(* Logix 5000 project; controller cal1632 1756-L62 rev 16.20; software revision 16.05; part 59 of 61 *)
(* tags used below, declared in another part *)
   AFI : BOOL;
   FAULT : BOOL;
   HMI : BOOL;
   p00_lin_timer_pre_0ms : DINT;
   p00_lin_timer_pre_1s : DINT;
   p00_lin_timer_pre_disc : DINT;
   p00_wac : Accumulator;   // Winder Accumulator
   p01_param_master_decel : REAL;
   p01r09 : routine;
   p01r09_pb_global_reset : BOOL;
   p01r12_master_ramped_speed : REAL;
   p01r13_line_running : BOOL;
   p01r13_line_slow_ramp : BOOL;
   p02_recipe_from_hmi : recipe;
   p29_di_wdr_a : BOOL;
   p29_param_acc_park_sp : REAL;   // Winder Accumulator Speed Trim Park Setpoint - Where the Carriage Sits [% of Stroke]
   p29r09_torque_mode : BOOL;
   p29r09_winder_a_active : BOOL;
   p29r09_winder_b_active : BOOL;
   p29r10 : routine;
   p29r10_request_run : BOOL;
   p29r11 : routine;
   p29r11_request_run : BOOL;
   p29r15_request_run : BOOL;
   p29r16_request_run : BOOL;
   p30_di_pin_1 : BOOL;
   p30_di_pin_2 : BOOL;
   p30_di_pin_3 : BOOL;
   p30_di_pin_4 : BOOL;
   p30_di_pin_5 : BOOL;
   p30_di_pin_6 : BOOL;
   p30_di_pin_7 : BOOL;
   p30_di_pin_8 : BOOL;
   p30_di_retraction_down_ls : BOOL;
   p30_di_retraction_up_ls : BOOL;
   p30_di_rotation_fault : BOOL;
   p30_do_retract_motion : BOOL;
   p30_do_rotation_fwd : BOOL;
   p30_do_rotation_rev : BOOL;
   p30r09_mode_close : BOOL;
   p30r09_mode_open : BOOL;
   p30r10 : routine;
   p30r10_motion_monitor_dwell : TIMER;
   p30r10_request_close : BOOL;
   p30r10_request_monitor : BOOL;
   p30r10_request_open : BOOL;
   p30r10_run_permissive : BOOL;
   p30r10_safety_pins_stowed : BOOL;
   p30r10_timer_fault : TIMER[4];
   p30r10_timer_warning : TIMER[4];
(* P30_Retraction_System, continued *)

ROUTINE R10_Retraction   (* ladder *)
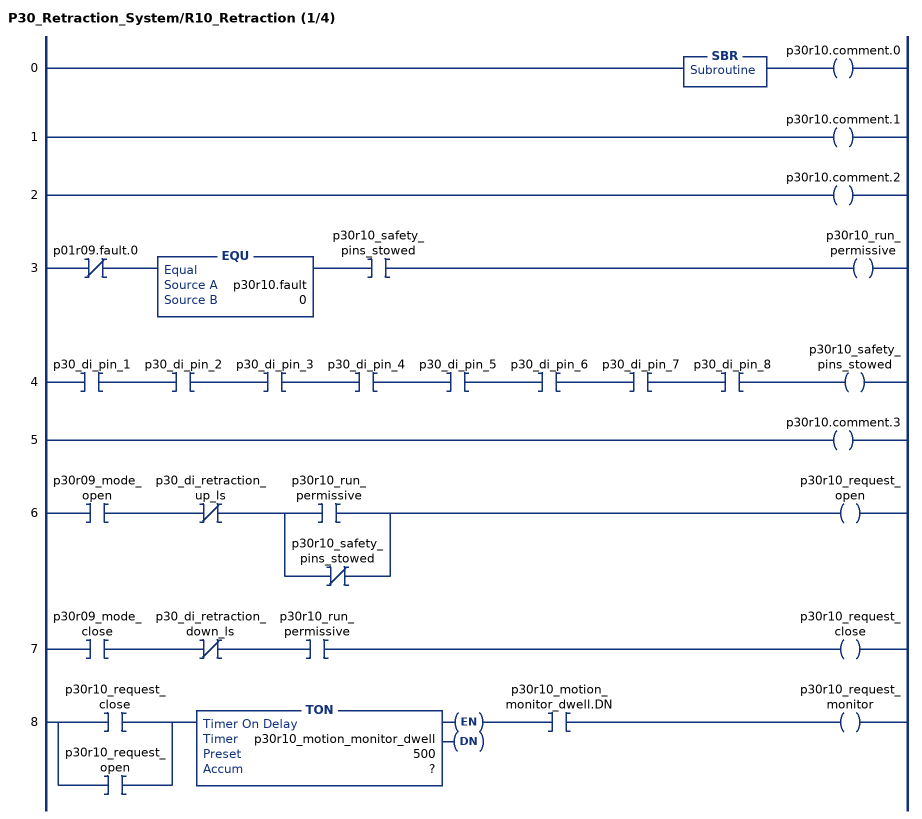
   0: SBR()OTE(p30r10.comment.0);
   1: OTE(p30r10.comment.1);
   2: OTE(p30r10.comment.2);
   3: XIO(p01r09.fault.0)EQU(p30r10.fault,0)XIC(p30r10_safety_pins_stowed)OTE(p30r10_run_permissive);
   4: XIC(p30_di_pin_1)XIC(p30_di_pin_2)XIC(p30_di_pin_3)XIC(p30_di_pin_4)XIC(p30_di_pin_5)XIC(p30_di_pin_6)XIC(p30_di_pin_7)XIC(p30_di_pin_8)OTE(p30r10_safety_pins_stowed);
   5: OTE(p30r10.comment.3);
   6: XIC(p30r09_mode_open)XIO(p30_di_retraction_up_ls)[XIC(p30r10_run_permissive) ,XIO(p30r10_safety_pins_stowed) ]OTE(p30r10_request_open);
   7: XIC(p30r09_mode_close)XIO(p30_di_retraction_down_ls)XIC(p30r10_run_permissive)OTE(p30r10_request_close);
   8: [XIC(p30r10_request_close) ,XIC(p30r10_request_open) ]TON(p30r10_motion_monitor_dwell,?,?)XIC(p30r10_motion_monitor_dwell.DN)OTE(p30r10_request_monitor);
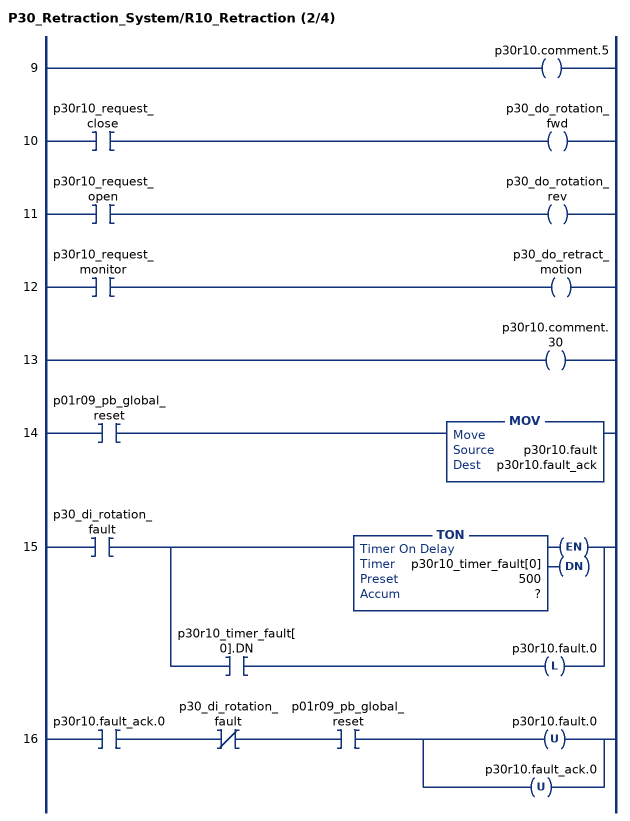
   9: OTE(p30r10.comment.5);
   10: XIC(p30r10_request_close)OTE(p30_do_rotation_fwd);
   11: XIC(p30r10_request_open)OTE(p30_do_rotation_rev);
   12: XIC(p30r10_request_monitor)OTE(p30_do_retract_motion);
   13: OTE(p30r10.comment.30);
   14: XIC(p01r09_pb_global_reset)MOV(p30r10.fault,p30r10.fault_ack);
   15: XIC(p30_di_rotation_fault)[TON(p30r10_timer_fault[0],?,?) ,XIC(p30r10_timer_fault[0].DN) OTL(p30r10.fault.0) ];
   16: XIC(p30r10.fault_ack.0)XIO(p30_di_rotation_fault)XIC(p01r09_pb_global_reset)[OTU(p30r10.fault.0) ,OTU(p30r10.fault_ack.0) ];
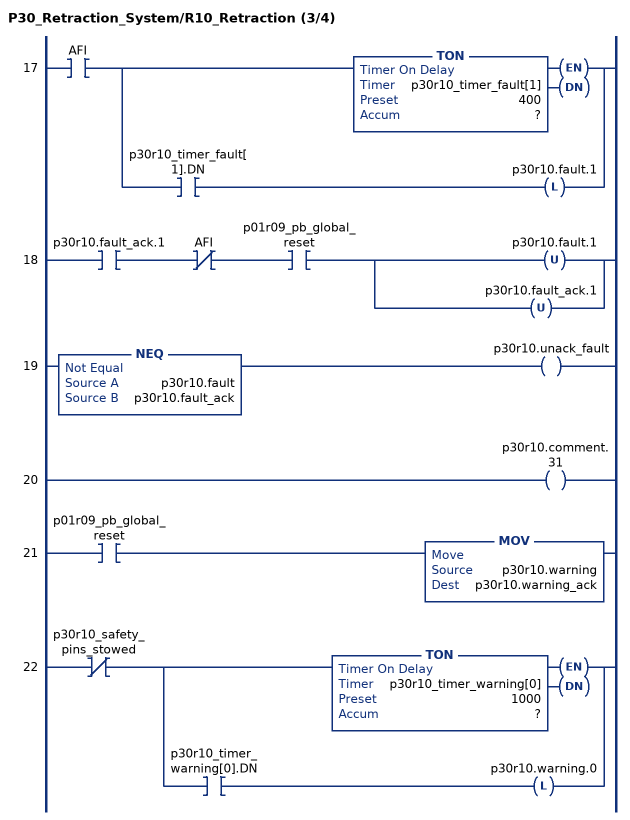
   17: XIC(AFI)[TON(p30r10_timer_fault[1],?,?) ,XIC(p30r10_timer_fault[1].DN) OTL(p30r10.fault.1) ];
   18: XIC(p30r10.fault_ack.1)XIO(AFI)XIC(p01r09_pb_global_reset)[OTU(p30r10.fault.1) ,OTU(p30r10.fault_ack.1) ];
   19: NEQ(p30r10.fault,p30r10.fault_ack)OTE(p30r10.unack_fault);
   20: OTE(p30r10.comment.31);
   21: XIC(p01r09_pb_global_reset)MOV(p30r10.warning,p30r10.warning_ack);
   22: XIO(p30r10_safety_pins_stowed)[TON(p30r10_timer_warning[0],?,?) ,XIC(p30r10_timer_warning[0].DN) OTL(p30r10.warning.0) ];
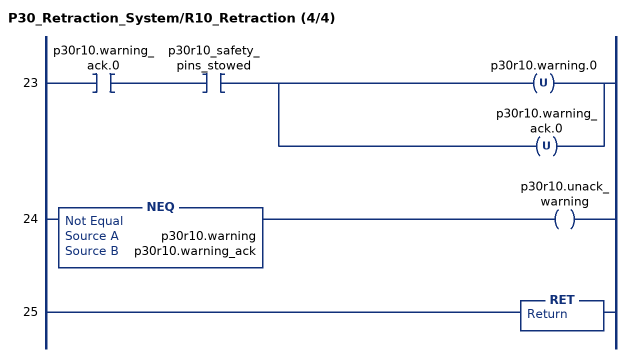
   23: XIC(p30r10.warning_ack.0)XIC(p30r10_safety_pins_stowed)[OTU(p30r10.warning.0) ,OTU(p30r10.warning_ack.0) ];
   24: NEQ(p30r10.warning,p30r10.warning_ack)OTE(p30r10.unack_warning);
   25: RET();
END_ROUTINE
END_PROGRAM

PROGRAM P31_WAC
// Winder Accumulator
VAR
   A00 : ALIAS FOR hmi_dint[0].0;
   A01 : ALIAS FOR hmi_dint[0].1;
   A02 : ALIAS FOR hmi_dint[0].2;
   A03 : ALIAS FOR hmi_dint[0].3;
   A04 : ALIAS FOR hmi_dint[0].4;
   A05 : ALIAS FOR hmi_dint[0].5;
   A06 : ALIAS FOR hmi_dint[0].6;
   A07 : ALIAS FOR hmi_dint[0].7;
   A08 : ALIAS FOR hmi_dint[0].8;
   A09 : ALIAS FOR hmi_dint[0].9;
   A10 : ALIAS FOR hmi_dint[0].10;
   A11 : ALIAS FOR hmi_dint[0].11;
   A12 : ALIAS FOR hmi_dint[0].12;
   A13 : ALIAS FOR hmi_dint[0].13;
   A14 : ALIAS FOR hmi_dint[0].14;
   A15 : ALIAS FOR hmi_dint[0].15;
   A16 : ALIAS FOR hmi_dint[0].16;
   A17 : ALIAS FOR hmi_dint[0].17;
   A18 : ALIAS FOR hmi_dint[0].18;
   A19 : ALIAS FOR hmi_dint[0].19;
   A20 : ALIAS FOR hmi_dint[0].20;
   A21 : ALIAS FOR hmi_dint[0].21;
   A22 : ALIAS FOR hmi_dint[0].22;
   A23 : ALIAS FOR hmi_dint[0].23;
   A24 : ALIAS FOR hmi_dint[0].24;
   A25 : ALIAS FOR hmi_dint[0].25;
   A26 : ALIAS FOR hmi_dint[0].26;
   A27 : ALIAS FOR hmi_dint[0].27;
   A28 : ALIAS FOR hmi_dint[0].28;
   A29 : ALIAS FOR hmi_dint[0].29;
   A30 : ALIAS FOR hmi_dint[0].30;
   A31 : ALIAS FOR hmi_dint[0].31;
   aaa_cjj_test_real1 : REAL;
   aaa_close_nip_from_feedroll : BOOL;
   acc_decel_reserve_pct : REAL;   // Accumulator Stroke Reserved for the Line Decel at the Present Line Speed [% of Stroke]
   acc_empty_limit : BOOL := 1;   // Accumulator Empty Limit
   acc_fill_status : DINT;
   acc_full_limit : BOOL;   // Accumulator Full Limit
   acc_norm_stop_pct : REAL := 60.0;   // Accumulator Normal Stop Threshold Computed - Full Limit Less Decel Reserve [% of Stroke]
   acc_position_last : REAL;
   acc_status : ALIAS FOR hmi_dint[13];
   accum_filling_on : ALIAS FOR hmi_dint[9].12;
   accum_holding_pressure_on : BOOL;   // Accumulator Holding Pressure Active
   accum_tension_pressure_on : BOOL := 1;   // Accumulator Tension Pressure Active
   accumulator_state : DINT := 33;   // Accumulator Sequence State Word
        .0   // Accumulator Sequence State One Step per Scan
        .1   // Accumulator Sequence State 1 Off
        .2   // Accumulator Sequence State 2 Control to Low Position
        .3   // Accumulator Sequence State 3 Fill Request
        .4   // Accumulator Sequence State 4 Fill to Full Position
        .5   // Accumulator Sequence State 5 Control to Upper Position
        .6   // Accumulator Sequence State 6 Payout Request
        .7   // Accumulator Sequence State 7 Lower Limit Reached
        .8   // Accumulator Sequence State 8
        .9   // Accumulator Sequence State 9
        .10   // Accumulator Sequence State 10
        .11   // Accumulator Sequence State 11
        .12   // Accumulator Sequence State 12
   add_sys_Acknowledge : sys_Acknowledge;   // Addon Acknowledge
   add_sys_filter_lpt : sys_Filter := (filter := 0.061195374, In_real := 0.061195374, Out_Real := 1.0);   // Addon Filter
   add_sys_Limit_Clamp : sys_Limit_Clamp := (max := 50.0);   // Addon System Limit Clamp
   add_sys_ramp : sys_Ramp := (IN_accel_rate := 29.0, IN_decel_rate := 200.0, IN_last_scan_s := 200.0, IN_target_setpoint := 0.05);   // Addon Ramp
   add_sys_scp : SYS_SCP := (Input := 29.0, Input_Max := 100.0, Output_Min := 4000.0, Output_Max := 20000.0, Output := 8640.0);   // Addon Scale with Parameters
   ai_lpt01_pct : REAL := 0.061195374;   // AI: Linear Position Transducer [%]
   ai_lpt01_raw : REAL := 5.086914;   // AI: Linear Position Transducer Unfiltered/Raw
   ai_pos01_pct_flt : REAL := 0.0667572;   // AI: Linear Position Transducer
   ai_ten01 : REAL;
   ai_tension : REAL;   // AI: Winder Accumulator Tension
   alarm_exists : ALIAS FOR hmi_dint[9].28;
   alm_ack : DINT[2];   // Accumulator Alarm Acknowledge Bits
   ao_prs01 : REAL := 0.4;   // AO: Pressure 1
   ao_prs02 : REAL := 29.0;   // AO: Pressure 2
   clamp_norm_stop : sys_Limit_Clamp;   // Accumulator Normal Stop Threshold Clamp
   control_to_empty : ALIAS FOR hmi_dint[9].13;
   di_high_limit : ALIAS FOR p00_io_winder:6:I.0;
   di_low_limit : ALIAS FOR p00_io_winder:5:I.5;
   di_pb_e_stop : ALIAS FOR p00_io_winder:5:I.15;
   di_pb_line_stop : ALIAS FOR p00_io_winder:5:I.7;
   di_ss_acc_on : ALIAS FOR p00_io_winder:5:I.6;
   di_ss_close_nip : ALIAS FOR p00_io_winder:5:I.14;
   di_ss_nip_auto : ALIAS FOR p00_io_winder:5:I.13;
   do_carriage_lift_sol : ALIAS FOR p00_io_winder:4:O.7;
   do_close_nip_sol : ALIAS FOR p00_io_winder:4:O.8;
   do_nip_illuminated_ss : ALIAS FOR p00_io_winder:4:O.6;
   empty_request : BOOL;   // Accumulator Empty Request
   enable_control : BOOL := 1;   // Accumulator - Enable Control
   filling_pressure : REAL;   // Accumulator Fill Pressure Tare + Tension + Fill PID Offset
   hmi_dint : DINT[20] := ([6] := 65504, [7] := 1, [9] := 8196, [11] := 5);
        [0].0   // A00 Emergency Stop
        [0].1   // A01
        [0].2   // A02
        [0].3   // A03
        [0].4   // A04 Accumulator Empty Limit
        [0].5   // A05 Accumulator Full Limit
        [0].6   // A06 Accumulator Nearly Empty Limit
        [0].7   // A07 Accumulator Nearly Full Limit
        [0].8   // A08 Accumulator Position Signal Fault
        [0].9   // A09
        [0].10   // A10
        [0].11   // A11
        [0].12   // A12
        [0].13   // A13
        [0].14   // A14
        [0].15   // A15 Tension Disabled
        [0].16   // A16
        [0].17   // A17
        [0].18   // A18
        [0].19   // A19
        [0].20   // A20
        [0].21   // A21
        [0].22   // A22
        [0].23   // A23
        [0].24   // A24
        [0].25   // A25
        [0].26   // A26
        [0].27   // A27
        [0].28   // A28
        [0].29   // A29
        [0].30   // A30
        [0].31   // A31
        [2].0   // W00 Nip Mode Warning
        [2].1   // W01 Accumulator Full - Line Stopped
        [2].2   // W02 Nip Selector Open - Accumulator On
        [2].3   // W03
        [2].4   // W04
        [2].5   // W05 Accumulator Off
        [2].6   // W06 Line Stop PB Pressed
        [2].7   // W07
        [2].8   // W08
        [2].9   // W09
        [2].10   // W10
        [2].11   // W11
        [2].12   // W12
        [2].13   // W13
        [2].14   // W14
        [2].15   // W15
        [2].16   // W16
        [2].17   // W17
        [2].18   // W18
        [2].19   // W19
        [2].20   // W20
        [2].21   // W21
        [2].22   // W22
        [2].23   // W23
        [2].24   // W24
        [2].25   // W25
        [2].26   // W26
        [2].27   // W27
        [2].28   // W28
        [2].29   // W29
        [2].30   // W30
        [2].31   // W31
        [4].10   // Accumulator PB: Enable Tension
        [7].0   // HMI DO: Accumulator On
        [7].1   // HMI DO: Close Nip
        [9].0   // Accumulator Sequence Request Reset
        [9].1   // Accumulator Sequence Request Fill
        [9].2   // Accumulator Accumulator On
        [9].7   // Accumulator Nip Close Request
        [9].8   // Accumulator Fill Pressure Request Position Control
        [9].10   // Accumlator Tension Request
        [9].12   // Accumulator FIlling Active
        [9].13   // Accumulator Control To Empty
        [9].15   // PID Manual Mode
        [9].28   // Accumulator Alarms Alarm Exists
        [9].29   // Accumulator Alarms Unacknowledged Alarm Exists
        [9].30   // Accumulator Warnings Warning Exists
        [9].31   // Accumulator Warnings Unacknowledged Warning Exists
        [13]   // Accumulator Status
        [15]   // Line Run Status
   hmi_pb_enable_tension : ALIAS FOR hmi_dint[4].10;
   IN_ai_lc01 : ALIAS FOR Local:3:I.Ch2Data;
   IN_ai_lpt01 : ALIAS FOR p00_io_oven:1:I.Ch4Data;
   line_run_status : ALIAS FOR hmi_dint[15];
   local_pb : DINT;
        .0   // Accumulator PB00
        .1   // Accumulator PB01
        .4   // Accumulator PB04: Enable Tension
        .30   // Accumulator PB: Stop Line
        .31   // Accumulator PB: Reset Zone
   lpt_raw_ok : BOOL := 1;   // Accumulator LPT Raw Signal In Range
   lpt_ref_pct : REAL;   // Accumulator LPT Frozen Detect Reference Position
   Me : ALIAS FOR p00_wac;
   nip_auto_open_request : BOOL := 1;   // Nip Auto Open Request
   nip_close_request : ALIAS FOR hmi_dint[9].7;
   nip_mode_auto : BOOL := 1;   // Nip Mode Auto
   nip_open_dwell : TIMER := (PRE := 2000);   // Nip Roll Open Dwell Payout must be established before the nip lets go
   nip_open_request : BOOL := 1;   // Nip Open Request
   nip_open_selected : BOOL;   // Nip Selector in OPEN Neither Auto nor Close
   oneshot : DINT;
   OUT_ao_prs01 : ALIAS FOR p00_io_winder:1:O.Ch3Data;
   OUT_ao_prs02 : ALIAS FOR p00_io_winder:1:O.Ch2Data;
   param_acc_capacity_ft : REAL := 10.0;   // Parameter Accumulator Web Capacity at Full Stroke 26 s at 23 fpm measured [ft]
   param_acc_full_clear_pct : REAL := 70.0;   // Parameter Accumulator Full Self-Clear the Line Stop Below This Position [% of Stroke]
   param_acc_full_stop_pct : REAL := 90.0;   // Parameter Accumulator Full Request Normal Line Stop Above This Position [% of Stroke]
   param_acc_handover_band_pct : REAL := 15.0;   // Parameter Accumulator Handover Band Stroke Over Which the Payout Boost Fades Out [% of Stroke]
   param_acc_handover_pct : REAL := 20.0;
   param_acc_low_pstn_sp : REAL;   // Parameter Accumulator Low Position Setpoint
   param_acc_low_tension_sp : REAL := 10.0;   // Parameter Accumulator Low Tension Setpoint
   param_acc_max_limit : REAL := 97.0;   // Parameter Accumulator High Max Limit
   param_acc_min_limit : REAL := 4.5;   // Parameter Accumulator Low Min Limimt
   param_acc_stop_hyst_pct : REAL := 20.0;   // Parameter Normal Stop Self-Clear Hysteresis Below the Threshold [% of Stroke]
   param_acc_stop_margin_pct : REAL := 5.0;   // Parameter Normal Stop Extra Margin Above the Decel Reserve [% of Stroke]
   param_accel_rate : REAL := 200.0;   // Parameter Acceleration Rate
   param_counter_prs : REAL := 0.4;   // Parameter Counter Pressure
   param_cv01_manual_sp : REAL := 7.0;
   param_decel_rate : REAL := 200.0;   // Parameter Decleration Rate
   param_empty_pct : REAL := 2.0;   // Parameter Empty Percent
   param_fill_SO : REAL := 70.0;   // Parameter FIll Pressure
   param_filter : REAL := 1.0;
   param_gain : REAL := 0.5;   // Parameter Gain
   param_high_ctrl_pct : REAL;   // Parameter High Control Position
   param_holding_pressure : REAL := 14.0;   // Parameter Carriage Holding Pressure
   param_low_ctrl_pct : REAL;   // Parameter Low Control Position
   param_lpt_frozen_ms : DINT := 30000;   // Parameter LPT Frozen Detect Dwell [ms]
   param_lpt_raw_max : DINT := 19000;   // Parameter LPT Raw Counts Upper Validity Limit
   param_lpt_raw_min : DINT := 200;   // Parameter LPT Raw Counts Lower Validity Limit
   param_max_counter_prs : REAL := 50.0;   // Parameter Max Counter Pressure
   param_min_counter_prs : REAL;   // Parameter Min Counter Pressure
   param_pid_kd : REAL := 0.0027322604;   // Parameter PID Kd
   param_pid_ki : REAL := 10.451622;   // Parameter PID Ki
   param_pid_kp : REAL := 0.7025812;   // Parameter PID Kp
   param_pid_process_type : DINT := 5;   // PIDE Process Type Selected by Autotune at the HMI
   param_press_offset : REAL := 83.0;   // Parameter Pressure Curve Offset Carriage weight term, vendor curve [lbf]
   param_press_slope_empty : REAL := 4.14;   // Parameter Pressure Curve Slope - EMPTYING Web Tension lb = slope x psi - offset [lb/psi]
   param_press_slope_fill : REAL := 3.75;   // Parameter Pressure Curve Slope - FILLING Web Tension lb = slope x psi - offset [lb/psi]
   param_sys_filter_lc01 : REAL;   // System Filter Parameter
   param_tare_pressure : REAL;   // Parameter Friction Trim Pressure Carriage Balanced - No Drift Up or Down Set at Installation
   payout_active : BOOL := 1;
   payout_pressure : REAL := 29.0;
   pb0 : ALIAS FOR hmi_dint[4];
   pb1 : ALIAS FOR hmi_dint[5];
   pb_acc_on : ALIAS FOR hmi_dint[9].2;
   pb_enable_tension : ALIAS FOR local_pb.4;
   pb_reset : ALIAS FOR local_pb.31;
   pb_stop_line : ALIAS FOR local_pb.30;
   pid_ctrl_cv : REAL := 100.0;   // PID Control CV
   pid_ctrl_pv : REAL := 0.061195374;   // PID Control PV
   pid_ctrl_sp : REAL := 10.0;   // PID Control SP
   pid_mode_manual : ALIAS FOR hmi_dint[9].15;
   PID_offset : REAL := 25.0;   // Position PID Offset
   pstn_should_move : BOOL;   // Accumulator Position Must Be Changing Filling or Paying Out
   rcp_tension_pressure : REAL := 29.282001;   // Recipe Accumulator Tension Pressure
   recipe_tension : ALIAS FOR p02_recipe_from_hmi.winder_tension_sp;
   request_fill : ALIAS FOR hmi_dint[9].1;
   selected_pressure : REAL := 29.0;   // Accumulator Selected Tension Pressure
   sys_filter : sys_Filter;   // System Filter
   task_scan_time : REAL := 0.05;   // Task Scan Time
   task_scan_time_dint : DINT := 50000;   // Task Scan
   tension_pressure : REAL := 35.0;
   tension_pressure1 : DINT;
   timer_alarm : TIMER[32] := ([4].ACC := 3000, [4].EN := 1, [4].DN := 1, [6].PRE := 1000, [6].ACC := 1001, [6].EN := 1, [6].DN := 1, [7].PRE := 3000, [11].PRE := 315000, [14].PRE := 12000, [24].PRE := 1000, [25].PRE := 1000, [26].PRE := 1000, [27].PRE := 1000, [28].PRE := 1000, [29].PRE := 1000, [30].PRE := 1200000, [31].EN := 1, [31].DN := 1);   // Accumulator Alarms Delay Timer
   timer_lpt_frozen : TIMER := (PRE := 30000);   // Accumulator LPT Frozen Detect Timer
   timer_nip_open_delay : TIMER := (PRE := 2000, ACC := 2000, EN := 1, DN := 1);   // Nip Open Dwell Timer
   timer_warning : TIMER[48] := ([0].PRE := 3000, [2].PRE := 400000, [3].PRE := 900000, [5].PRE := 3000, [7].PRE := 3000, [8].PRE := 3000, [9].PRE := 3000, [11].PRE := 2500, [12].PRE := 2500, [13].PRE := 10000, [14].PRE := 10000, [15].PRE := 10000, [24].PRE := 15000, [24].ACC := 15001, [24].EN := 1, [24].DN := 1, [32].PRE := 3000, [33].PRE := 3000, [34].PRE := 3000, [35].PRE := 3000, [36].PRE := 3000, [37].PRE := 3000, [38].PRE := 3000, [39].PRE := 3000, [40].PRE := 3000, [41].PRE := 3000);   // Accumulator Warning Delay
   unack_alarm : ALIAS FOR hmi_dint[9].29;
   unack_warning : ALIAS FOR hmi_dint[9].31;
   use_auto_tune_gains : BOOL;   // Tension PIDE Use Auto Tune Values
   W00 : ALIAS FOR hmi_dint[2].0;
   W01 : ALIAS FOR hmi_dint[2].1;
   W02 : ALIAS FOR hmi_dint[2].2;
   W03 : ALIAS FOR hmi_dint[2].3;
   W04 : ALIAS FOR hmi_dint[2].4;
   W05 : ALIAS FOR hmi_dint[2].5;
   W06 : ALIAS FOR hmi_dint[2].6;
   W07 : ALIAS FOR hmi_dint[2].7;
   W08 : ALIAS FOR hmi_dint[2].8;
   W09 : ALIAS FOR hmi_dint[2].9;
   W10 : ALIAS FOR hmi_dint[2].10;
   W11 : ALIAS FOR hmi_dint[2].11;
   W12 : ALIAS FOR hmi_dint[2].12;
   W13 : ALIAS FOR hmi_dint[2].13;
   W14 : ALIAS FOR hmi_dint[2].14;
   W15 : ALIAS FOR hmi_dint[2].15;
   wac_calc_tension_pressure : REAL;   // Winder Accumulator Calulated Tension Pressure
   wac_empty : BOOL := 1;
   wac_empty_stop : BOOL;   // Accumulator Empty with No Winder Running Normal Line Stop Requested Self-Clearing
   wac_full_stop : BOOL;   // Accumulator Full - Normal Line Stop Requested Self-Clearing, No Reset Required
   wac_nearly_empty : BOOL := 1;
   wac_tension_pressure : REAL;   // Winder Accumulator Tare + Web Tension Pressure Carriage Holds Position at Commanded Tension
   warning_exists : ALIAS FOR hmi_dint[9].30;
   winder_running : BOOL := 1;   // Winder Running
   wrn_ack : DINT[2];   // Accumulator Warning Acknowledge Bits
   zzz_rate : REAL;
END_VAR

ROUTINE R00_Main   (* ladder *)
// Winder Accumulator
// Main
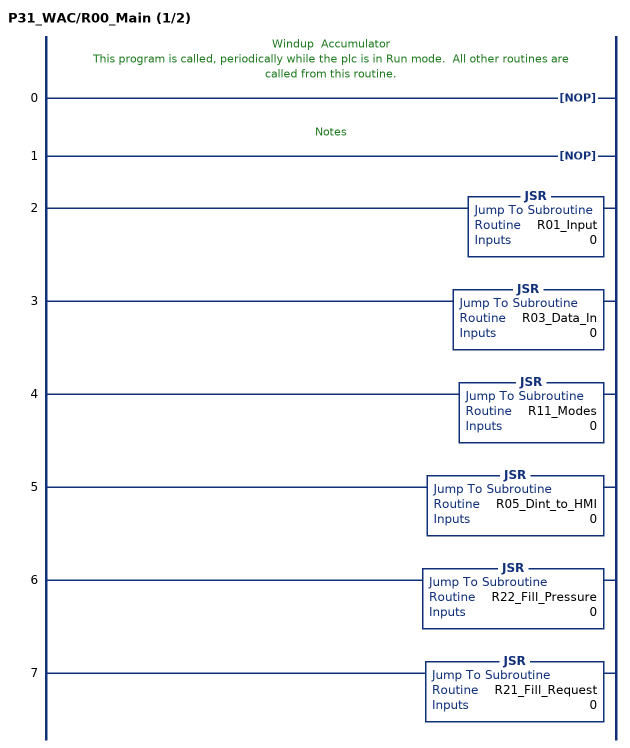
   // Windup  Accumulator
   // This program is called, periodically while the plc is in Run mode.  All other routines are called from this routine.
   0: NOP();
   // Notes
   1: NOP();
   2: JSR(R01_Input,0);
   3: JSR(R03_Data_In,0);
   4: JSR(R11_Modes,0);
   5: JSR(R05_Dint_to_HMI,0);
   6: JSR(R22_Fill_Pressure,0);
   7: JSR(R21_Fill_Request,0);
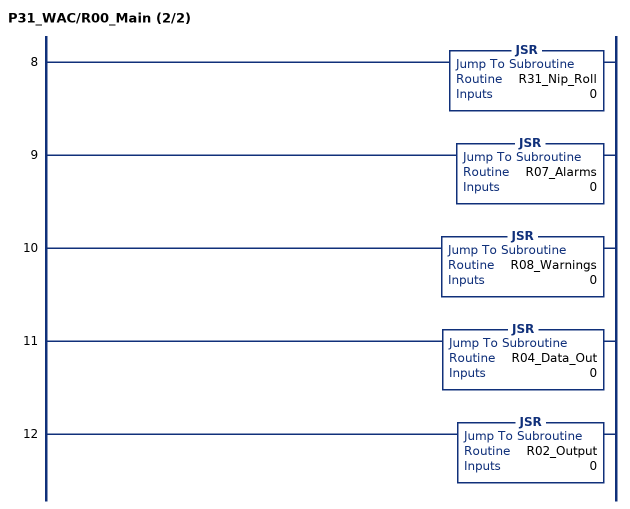
   8: JSR(R31_Nip_Roll,0);
   9: JSR(R07_Alarms,0);
   10: JSR(R08_Warnings,0);
   11: JSR(R04_Data_Out,0);
   12: JSR(R02_Output,0);
END_ROUTINE

ROUTINE R01_Input   (* ladder *)
// Windup Accumulator
// Input
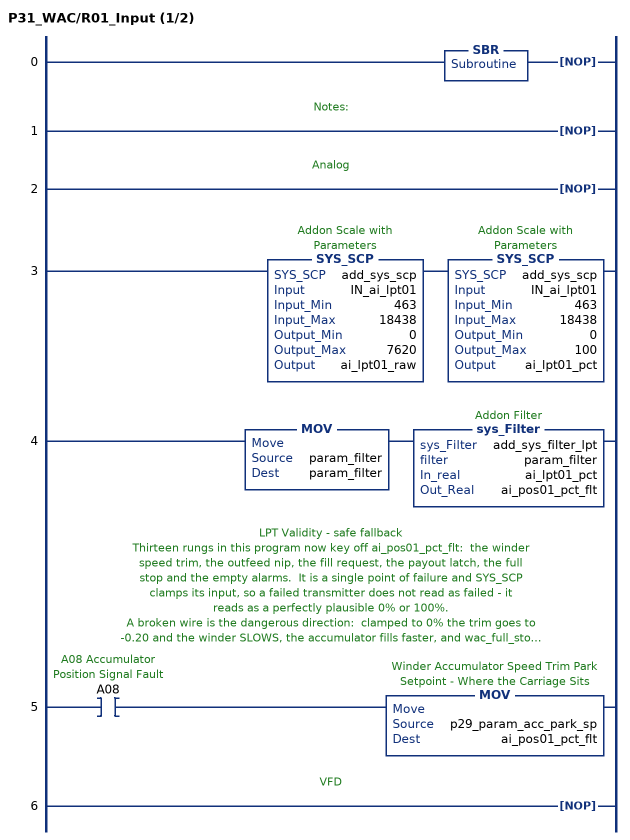
   0: SBR()NOP();
   // Notes:
   1: NOP();
   // Analog
   2: NOP();
   3: SYS_SCP(add_sys_scp,IN_ai_lpt01,463,18438,0,7620,ai_lpt01_raw)SYS_SCP(add_sys_scp,IN_ai_lpt01,463,18438,0,100,ai_lpt01_pct);
   4: MOV(param_filter,param_filter)sys_Filter(add_sys_filter_lpt,param_filter,ai_lpt01_pct,ai_pos01_pct_flt);
   // LPT Validity - safe fallback
   // Thirteen rungs in this program now key off ai_pos01_pct_flt:  the winder
   // speed trim, the outfeed nip, the fill request, the payout latch, the full
   // stop and the empty alarms.  It is a single point of failure and SYS_SCP
   // clamps its input, so a failed transmitter does not read as failed - it
   // reads as a perfectly plausible 0% or 100%.
   // A broken wire is the dangerous direction:  clamped to 0% the trim goes to
   // -0.20 and the winder SLOWS, the accumulator fills faster, and wac_full_stop
   // never trips because position reads empty.  Only di_high_limit would catch
   // it, at the mechanical stop.
   // So on A08 the position is forced to the park setpoint.  The trim then
   // computes zero and the winder tracks line speed, the nip stays open, and no
   // spurious full or empty is raised.  di_high_limit remains the hard backstop.
   // ai_lpt01_pct keeps the unfiltered reading for diagnosis on the HMI.
   // Rev 20260825 a09
   5: XIC(A08)MOV(p29_param_acc_park_sp,ai_pos01_pct_flt);
   // VFD
   6: NOP();
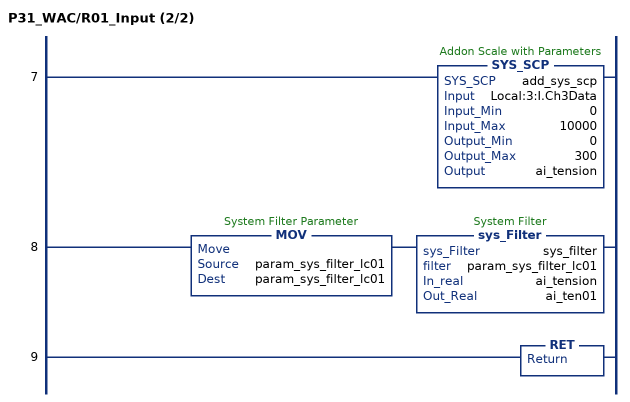
   7: SYS_SCP(add_sys_scp,Local:3:I.Ch3Data,0,10000,0,300,ai_tension);
   8: MOV(param_sys_filter_lc01,param_sys_filter_lc01)sys_Filter(sys_filter,param_sys_filter_lc01,ai_tension,ai_ten01);
   9: RET();
END_ROUTINE

ROUTINE R02_Output   (* ladder *)
// Windup Accumulator
// Output
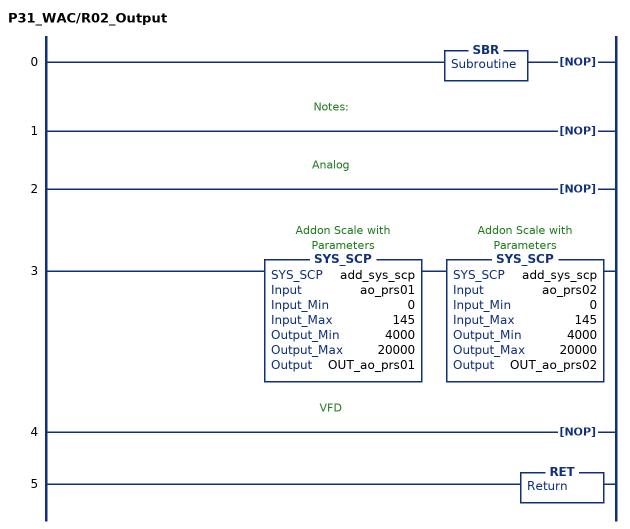
   0: SBR()NOP();
   // Notes:
   1: NOP();
   // Analog
   2: NOP();
   3: SYS_SCP(add_sys_scp,ao_prs01,0,145,4000,20000,OUT_ao_prs01)SYS_SCP(add_sys_scp,ao_prs02,0,145,4000,20000,OUT_ao_prs02);
   // VFD
   4: NOP();
   5: RET();
END_ROUTINE

ROUTINE R03_Data_In   (* ladder *)
// Windup Accumulator
// Data In
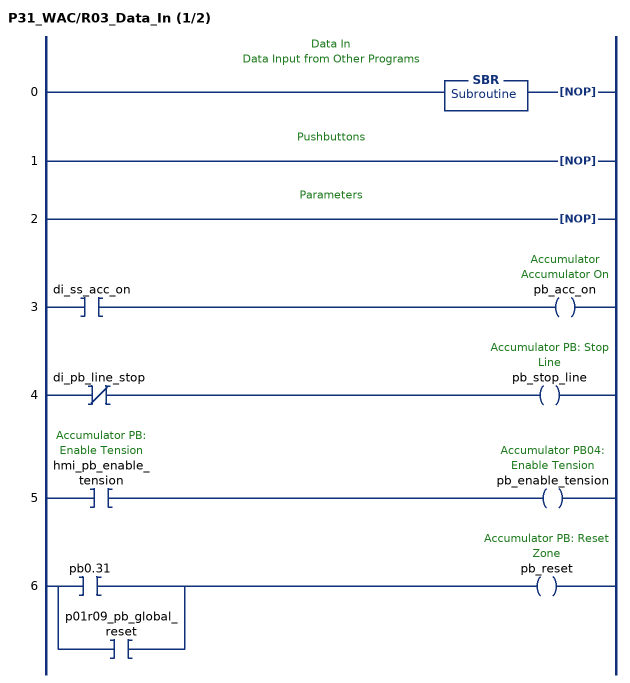
   // Data In
   // Data Input from Other Programs
   0: SBR()NOP();
   // Pushbuttons
   1: NOP();
   // Parameters
   2: NOP();
   3: XIC(di_ss_acc_on)OTE(pb_acc_on);
   4: XIO(di_pb_line_stop)OTE(pb_stop_line);
   5: XIC(hmi_pb_enable_tension)OTE(pb_enable_tension);
   6: [XIC(pb0.31) ,XIC(p01r09_pb_global_reset) ]OTE(pb_reset);
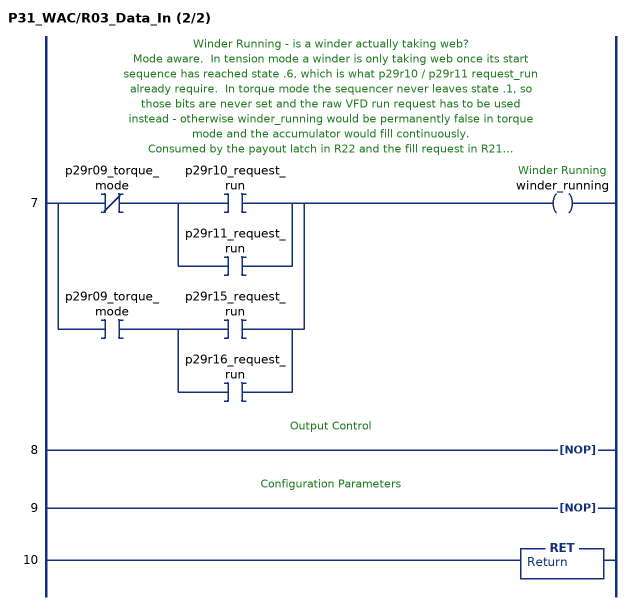
   // Winder Running - is a winder actually taking web?
   // Mode aware.  In tension mode a winder is only taking web once its start
   // sequence has reached state .6, which is what p29r10 / p29r11 request_run
   // already require.  In torque mode the sequencer never leaves state .1, so
   // those bits are never set and the raw VFD run request has to be used
   // instead - otherwise winder_running would be permanently false in torque
   // mode and the accumulator would fill continuously.
   // Consumed by the payout latch in R22 and the fill request in R21.
   // Rev 20260820 a02
   7: [XIO(p29r09_torque_mode) [XIC(p29r10_request_run) ,XIC(p29r11_request_run) ] ,XIC(p29r09_torque_mode) [XIC(p29r15_request_run) ,XIC(p29r16_request_run) ] ]OTE(winder_running);
   // Output Control
   8: NOP();
   // Configuration Parameters
   9: NOP();
   10: RET();
END_ROUTINE

ROUTINE R04_Data_Out   (* ladder *)
// Windup Accumulator
// Data Out
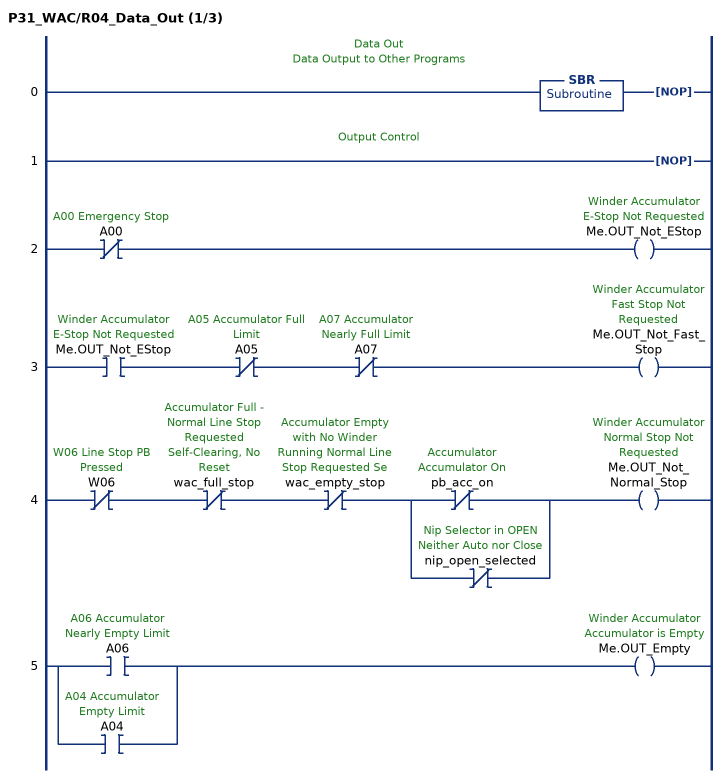
   // Data Out
   // Data Output to Other Programs
   0: SBR()NOP();
   // Output Control
   1: NOP();
   2: XIO(A00)OTE(Me.OUT_Not_EStop);
   3: XIC(Me.OUT_Not_EStop)XIO(A05)XIO(A07)OTE(Me.OUT_Not_Fast_Stop);
   4: XIO(W06)XIO(wac_full_stop)XIO(wac_empty_stop)[XIO(pb_acc_on) ,XIO(nip_open_selected) ]OTE(Me.OUT_Not_Normal_Stop);
   5: [XIC(A06) ,XIC(A04) ]OTE(Me.OUT_Empty);
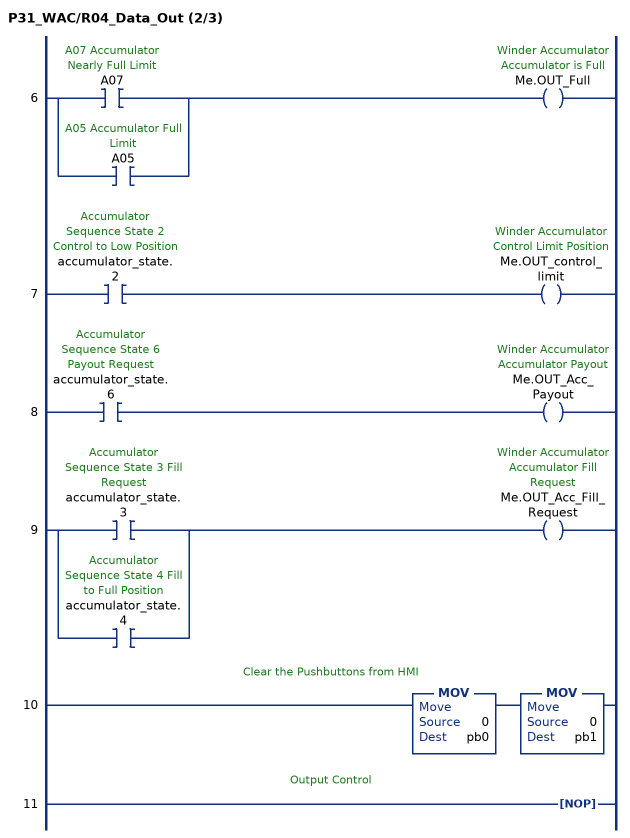
   6: [XIC(A07) ,XIC(A05) ]OTE(Me.OUT_Full);
   7: XIC(accumulator_state.2)OTE(Me.OUT_control_limit);
   8: XIC(accumulator_state.6)OTE(Me.OUT_Acc_Payout);
   9: [XIC(accumulator_state.3) ,XIC(accumulator_state.4) ]OTE(Me.OUT_Acc_Fill_Request);
   // Clear the Pushbuttons from HMI
   10: MOV(0,pb0)MOV(0,pb1);
   // Output Control
   11: NOP();
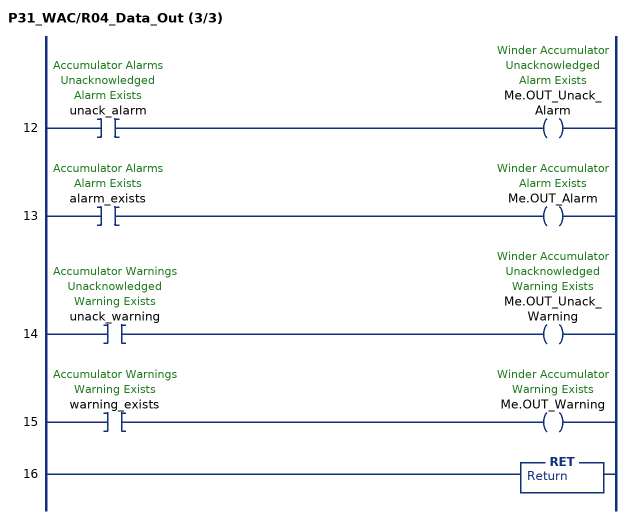
   12: XIC(unack_alarm)OTE(Me.OUT_Unack_Alarm);
   13: XIC(alarm_exists)OTE(Me.OUT_Alarm);
   14: XIC(unack_warning)OTE(Me.OUT_Unack_Warning);
   15: XIC(warning_exists)OTE(Me.OUT_Warning);
   16: RET();
END_ROUTINE

ROUTINE R05_Dint_to_HMI   (* ladder *)
// Windup  Accumulator
// Dint to HMI
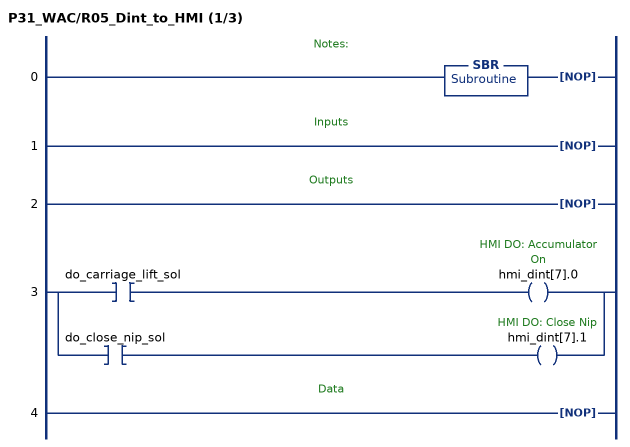
   // Notes:
   0: SBR()NOP();
   // Inputs
   1: NOP();
   // Outputs
   2: NOP();
   3: [XIC(do_carriage_lift_sol) OTE(hmi_dint[7].0) ,XIC(do_close_nip_sol) OTE(hmi_dint[7].1) ];
   // Data
   4: NOP();
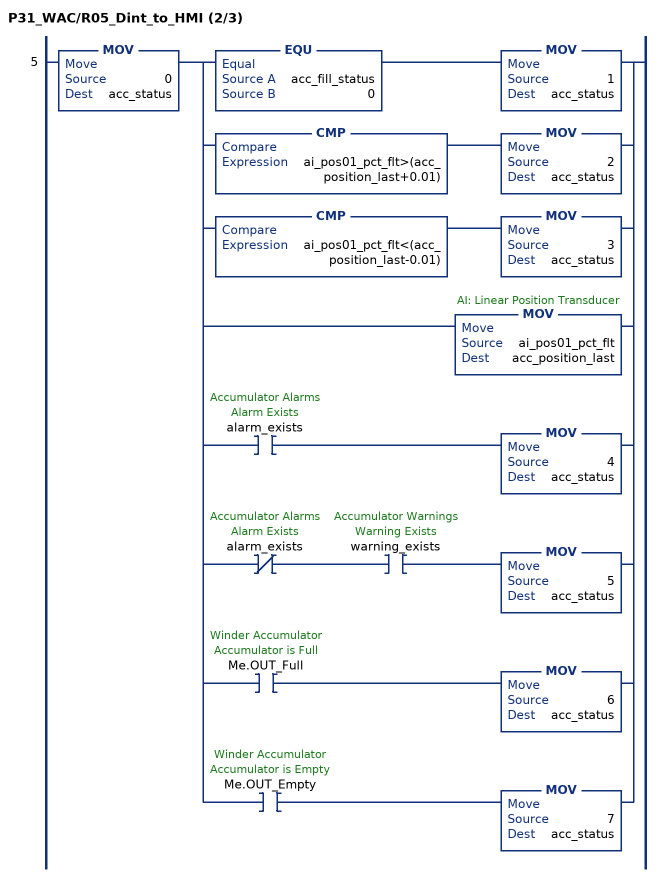
   5: MOV(0,acc_status)[EQU(acc_fill_status,0) MOV(1,acc_status) ,CMP(ai_pos01_pct_flt>(acc_position_last+0.01)) MOV(2,acc_status) ,CMP(ai_pos01_pct_flt<(acc_position_last-0.01)) MOV(3,acc_status) ,MOV(ai_pos01_pct_flt,acc_position_last) ,XIC(alarm_exists) MOV(4,acc_status) ,XIO(alarm_exists) XIC(warning_exists) MOV(5,acc_status) ,XIC(Me.OUT_Full) MOV(6,acc_status) ,XIC(Me.OUT_Empty) MOV(7,acc_status) ];
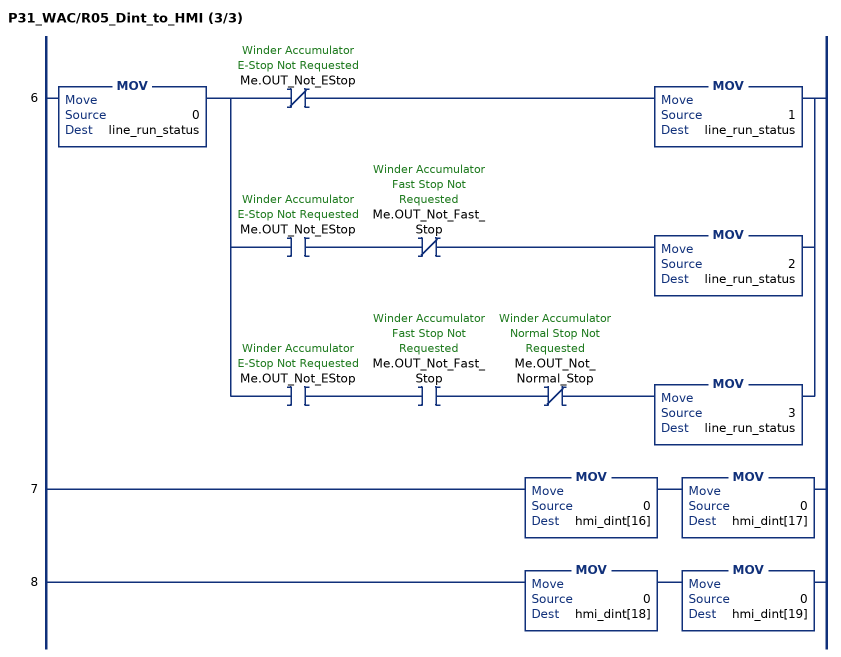
   6: MOV(0,line_run_status)[XIO(Me.OUT_Not_EStop) MOV(1,line_run_status) ,XIC(Me.OUT_Not_EStop) XIO(Me.OUT_Not_Fast_Stop) MOV(2,line_run_status) ,XIC(Me.OUT_Not_EStop) XIC(Me.OUT_Not_Fast_Stop) XIO(Me.OUT_Not_Normal_Stop) MOV(3,line_run_status) ];
   7: MOV(0,hmi_dint[16])MOV(0,hmi_dint[17]);
   8: MOV(0,hmi_dint[18])MOV(0,hmi_dint[19]);
END_ROUTINE

ROUTINE R07_Alarms   (* ladder *)
// Windup Accumulator
// Alarms
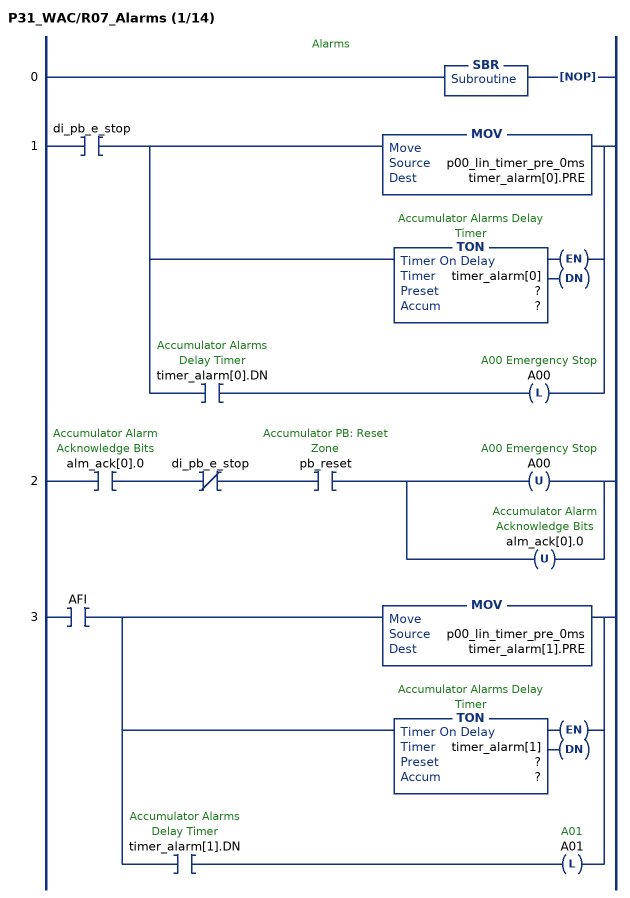
   // Alarms
   0: SBR()NOP();
   1: XIC(di_pb_e_stop)[MOV(p00_lin_timer_pre_0ms,timer_alarm[0].PRE) ,TON(timer_alarm[0],?,?) ,XIC(timer_alarm[0].DN) OTL(A00) ];
   2: XIC(alm_ack[0].0)XIO(di_pb_e_stop)XIC(pb_reset)[OTU(A00) ,OTU(alm_ack[0].0) ];
   3: XIC(AFI)[MOV(p00_lin_timer_pre_0ms,timer_alarm[1].PRE) ,TON(timer_alarm[1],?,?) ,XIC(timer_alarm[1].DN) OTL(A01) ];
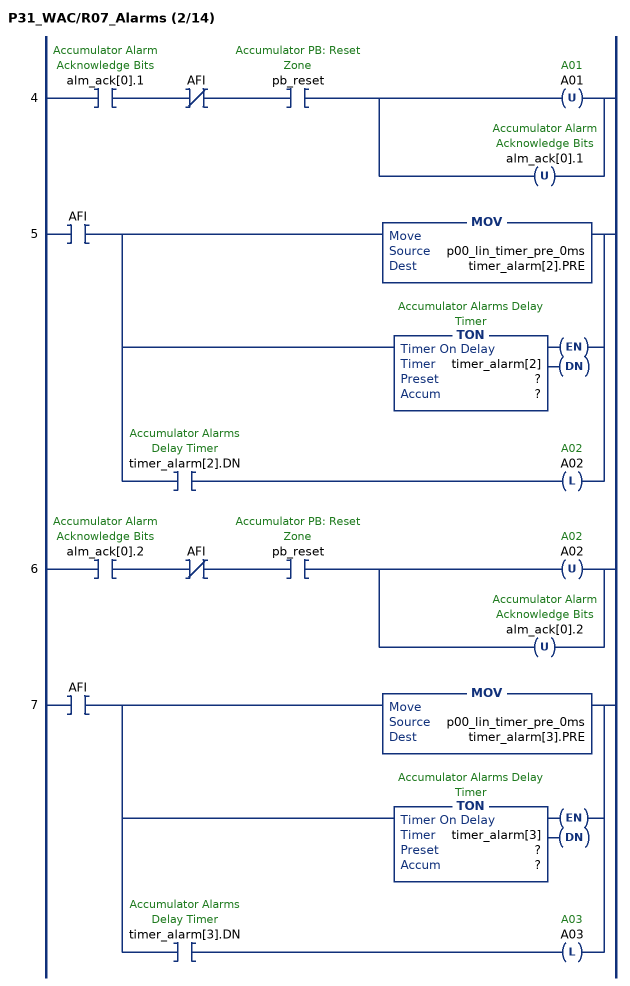
   4: XIC(alm_ack[0].1)XIO(AFI)XIC(pb_reset)[OTU(A01) ,OTU(alm_ack[0].1) ];
   5: XIC(AFI)[MOV(p00_lin_timer_pre_0ms,timer_alarm[2].PRE) ,TON(timer_alarm[2],?,?) ,XIC(timer_alarm[2].DN) OTL(A02) ];
   6: XIC(alm_ack[0].2)XIO(AFI)XIC(pb_reset)[OTU(A02) ,OTU(alm_ack[0].2) ];
   7: XIC(AFI)[MOV(p00_lin_timer_pre_0ms,timer_alarm[3].PRE) ,TON(timer_alarm[3],?,?) ,XIC(timer_alarm[3].DN) OTL(A03) ];
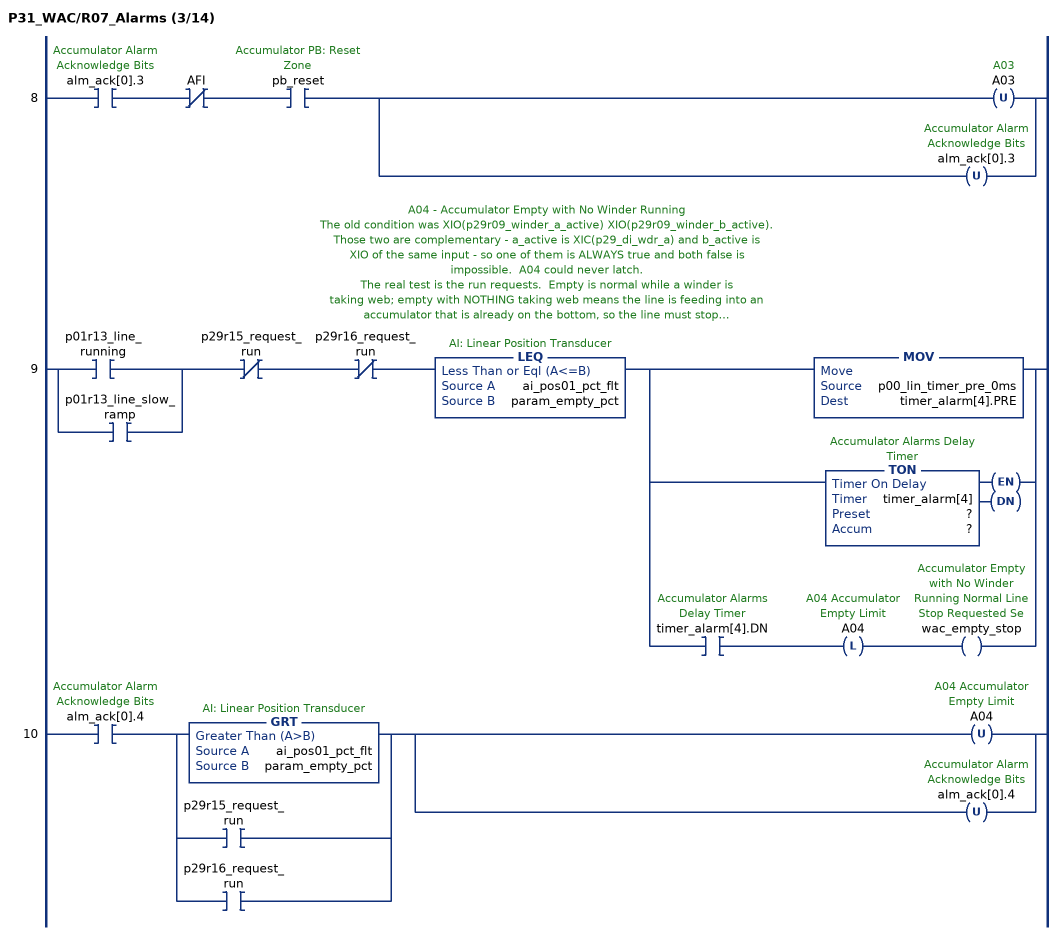
   8: XIC(alm_ack[0].3)XIO(AFI)XIC(pb_reset)[OTU(A03) ,OTU(alm_ack[0].3) ];
   // A04 - Accumulator Empty with No Winder Running
   // The old condition was XIO(p29r09_winder_a_active) XIO(p29r09_winder_b_active).
   // Those two are complementary - a_active is XIC(p29_di_wdr_a) and b_active is
   // XIO of the same input - so one of them is ALWAYS true and both false is
   // impossible.  A04 could never latch.
   // The real test is the run requests.  Empty is normal while a winder is
   // taking web; empty with NOTHING taking web means the line is feeding into an
   // accumulator that is already on the bottom, so the line must stop.
   // Gated on the line actually moving, with the standard 3 s dwell, so the
   // moment at line start - accumulator empty, winder not yet up - does not
   // trip it.
   // wac_empty_stop is the non-latching line stop, mirroring wac_full_stop.  A04
   // is the annunciation and still needs an acknowledge.
   // Rev 20260825 a16
   9: [XIC(p01r13_line_running) ,XIC(p01r13_line_slow_ramp) ]XIO(p29r15_request_run)XIO(p29r16_request_run)LEQ(ai_pos01_pct_flt,param_empty_pct)[MOV(p00_lin_timer_pre_0ms,timer_alarm[4].PRE) ,TON(timer_alarm[4],?,?) ,XIC(timer_alarm[4].DN) OTL(A04) OTE(wac_empty_stop) ];
   10: XIC(alm_ack[0].4)[GRT(ai_pos01_pct_flt,param_empty_pct) ,XIC(p29r15_request_run) ,XIC(p29r16_request_run) ][OTU(A04) ,OTU(alm_ack[0].4) ];
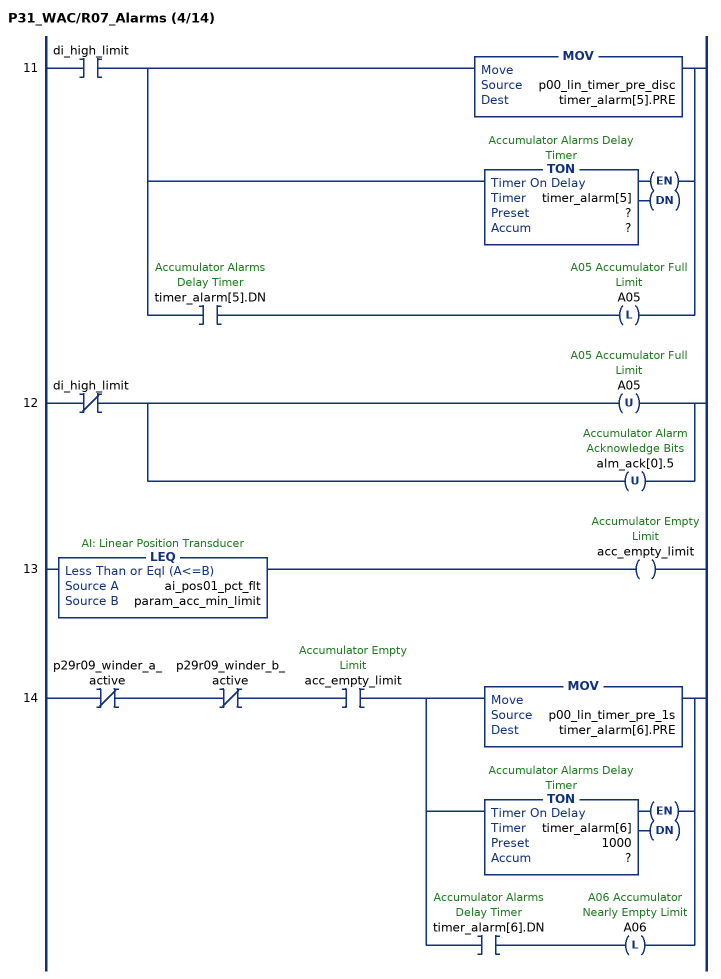
   11: XIC(di_high_limit)[MOV(p00_lin_timer_pre_disc,timer_alarm[5].PRE) ,TON(timer_alarm[5],?,?) ,XIC(timer_alarm[5].DN) OTL(A05) ];
   12: XIO(di_high_limit)[OTU(A05) ,OTU(alm_ack[0].5) ];
   13: LEQ(ai_pos01_pct_flt,param_acc_min_limit)OTE(acc_empty_limit);
   14: XIO(p29r09_winder_a_active)XIO(p29r09_winder_b_active)XIC(acc_empty_limit)[MOV(p00_lin_timer_pre_1s,timer_alarm[6].PRE) ,TON(timer_alarm[6],?,?) ,XIC(timer_alarm[6].DN) OTL(A06) ];
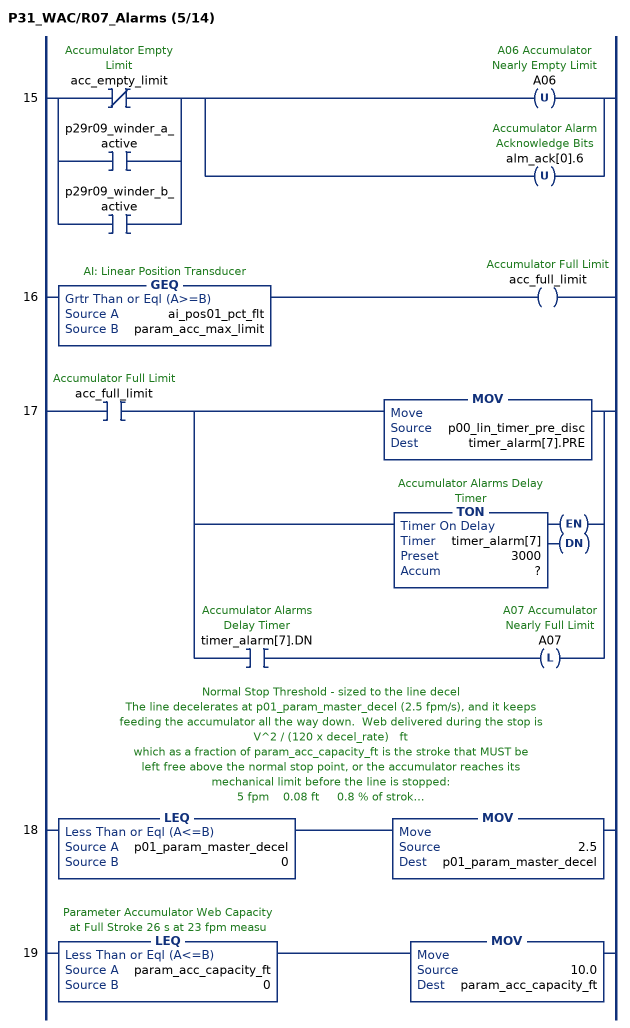
   15: [XIO(acc_empty_limit) ,XIC(p29r09_winder_a_active) ,XIC(p29r09_winder_b_active) ][OTU(A06) ,OTU(alm_ack[0].6) ];
   16: GEQ(ai_pos01_pct_flt,param_acc_max_limit)OTE(acc_full_limit);
   17: XIC(acc_full_limit)[MOV(p00_lin_timer_pre_disc,timer_alarm[7].PRE) ,TON(timer_alarm[7],?,?) ,XIC(timer_alarm[7].DN) OTL(A07) ];
   // Normal Stop Threshold - sized to the line decel
   // The line decelerates at p01_param_master_decel (2.5 fpm/s), and it keeps
   // feeding the accumulator all the way down.  Web delivered during the stop is
   //      V^2 / (120 x decel_rate)   ft
   // which as a fraction of param_acc_capacity_ft is the stroke that MUST be
   // left free above the normal stop point, or the accumulator reaches its
   // mechanical limit before the line is stopped:
   //       5 fpm    0.08 ft     0.8 % of stroke
   //      10 fpm    0.33 ft     3.3 %
   //      15 fpm    0.75 ft     7.5 %
   //      23 fpm    1.76 ft    17.6 %
   //      30 fpm    3.00 ft    30.0 %
   // The old fixed 90% left only 7% of stroke, which is only enough below about
   // 14 fpm.  Above that the line could not stop before the hard limit and the
   // fast stop always fired instead - which is exactly the steep stop this is
   // meant to avoid.
   // A fixed lower threshold would fix 30 fpm but throw away a third of the
   // accumulator at 5 fpm, where the decel needs almost nothing.  So the reserve
   // is computed from the present line speed instead, and the threshold floats
   // with it - the full accumulator is available at creep, the protection is
   // there at full speed.
   // Clamped between param_acc_handover_pct and param_acc_max_limit so a bad
   // speed or decel value can never push it outside the stroke.
   // Rev 20260825 a10
   18: LEQ(p01_param_master_decel,0)MOV(2.5,p01_param_master_decel);
   19: LEQ(param_acc_capacity_ft,0)MOV(10.0,param_acc_capacity_ft);
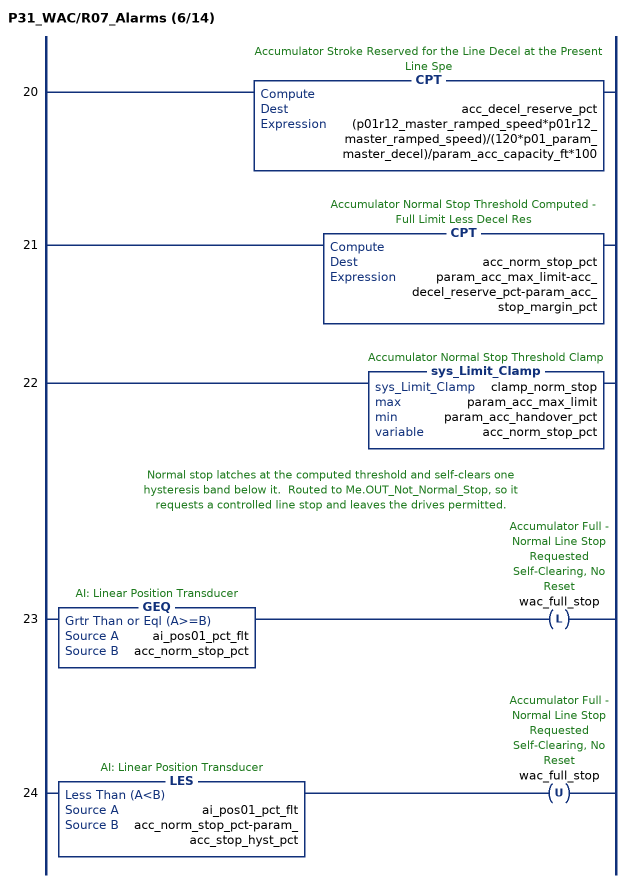
   20: CPT(acc_decel_reserve_pct,(p01r12_master_ramped_speed*p01r12_master_ramped_speed)/(120*p01_param_master_decel)/param_acc_capacity_ft*100);
   21: CPT(acc_norm_stop_pct,param_acc_max_limit-acc_decel_reserve_pct-param_acc_stop_margin_pct);
   22: sys_Limit_Clamp(clamp_norm_stop,param_acc_max_limit,param_acc_handover_pct,acc_norm_stop_pct);
   // Normal stop latches at the computed threshold and self-clears one
   // hysteresis band below it.  Routed to Me.OUT_Not_Normal_Stop, so it
   // requests a controlled line stop and leaves the drives permitted.
   23: GEQ(ai_pos01_pct_flt,acc_norm_stop_pct)OTL(wac_full_stop);
   24: LES(ai_pos01_pct_flt,acc_norm_stop_pct-param_acc_stop_hyst_pct)OTU(wac_full_stop);
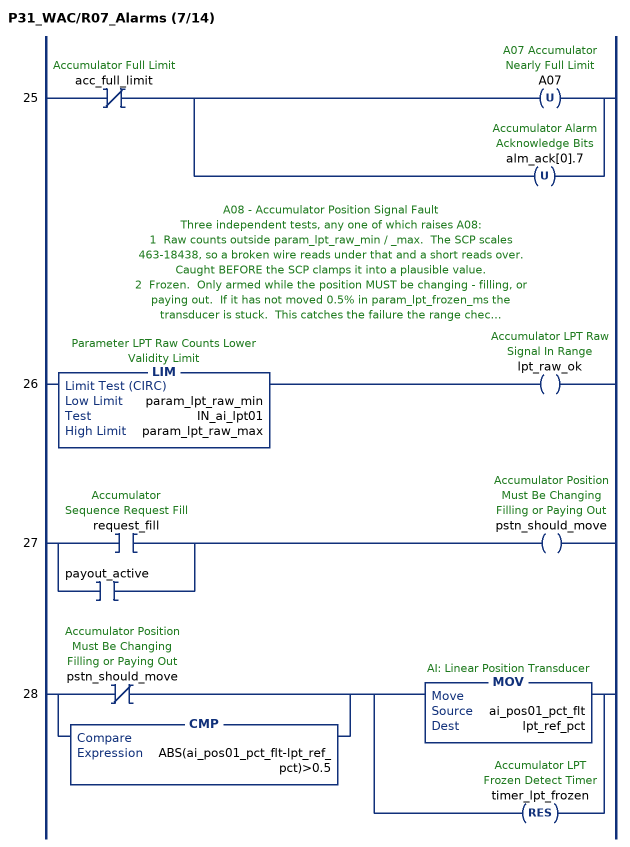
   25: XIO(acc_full_limit)[OTU(A07) ,OTU(alm_ack[0].7) ];
   // A08 - Accumulator Position Signal Fault
   // Three independent tests, any one of which raises A08:
   //   1  Raw counts outside param_lpt_raw_min / _max.  The SCP scales
   //      463-18438, so a broken wire reads under that and a short reads over.
   //      Caught BEFORE the SCP clamps it into a plausible value.
   //   2  Frozen.  Only armed while the position MUST be changing - filling, or
   //      paying out.  If it has not moved 0.5% in param_lpt_frozen_ms the
   //      transducer is stuck.  This catches the failure the range check
   //      cannot:  a signal that is in band but no longer tracking.
   //   3  Disagreement with di_high_limit - the discrete says full while the
   //      analog says it is below the full-stop threshold.  One of them lies.
   // Not self-clearing.  A sensor fault should be acknowledged deliberately,
   // unlike the process alarms A05 and A07.
   // Rev 20260825 a09
   26: LIM(param_lpt_raw_min,IN_ai_lpt01,param_lpt_raw_max)OTE(lpt_raw_ok);
   27: [XIC(request_fill) ,XIC(payout_active) ]OTE(pstn_should_move);
   28: [XIO(pstn_should_move) ,CMP(ABS(ai_pos01_pct_flt-lpt_ref_pct)>0.5) ][MOV(ai_pos01_pct_flt,lpt_ref_pct) ,RES(timer_lpt_frozen) ];
